PROGRAM P5_04_Trends
VAR
END_VAR

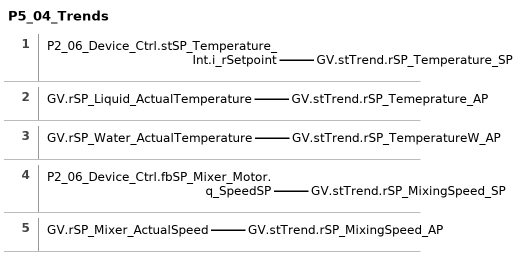
// NETWORK 1
GV.stTrend.rSP_Temperature_SP := P2_06_Device_Ctrl.stSP_Temperature_Int.i_rSetpoint;

// NETWORK 2
GV.stTrend.rSP_Temeprature_AP := GV.rSP_Liquid_ActualTemperature;

// NETWORK 3
GV.stTrend.rSP_TemperatureW_AP := GV.rSP_Water_ActualTemperature;

// NETWORK 4
GV.stTrend.rSP_MixingSpeed_SP := P2_06_Device_Ctrl.fbSP_Mixer_Motor.q_SpeedSP;

// NETWORK 5
GV.stTrend.rSP_MixingSpeed_AP := GV.rSP_Mixer_ActualSpeed;

END_PROGRAM

(* stored: Version 1.1.0.1, ProductVersion 3.1.4024.12
   POU P5_04_Trends: Id {f64f1721-1ac7-47fb-a84a-7efa6f3bea7a}, SpecialFunc None *)
